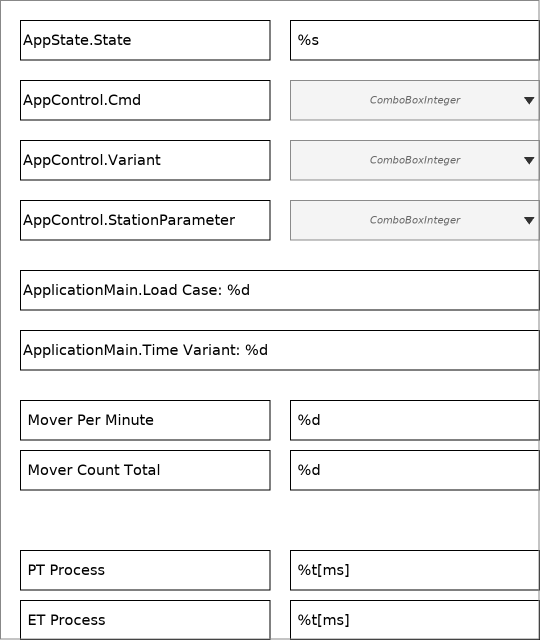
VISUALIZATION APP_CONTROL  // 540x640
    Rectangle (20,270 520x40), "ApplicationMain.Load Case: %d", text variable: GVL_APPLICATION.ApplicationMain._nLoadCase
        OnMouseClick: write the text variable via VisuDialogs.Numpad, min 0, max 2
    Rectangle (20,330 520x40), "ApplicationMain.Time Variant: %d", text variable: GVL_APPLICATION.ApplicationMain._nTimeVariant
        OnMouseClick: write the text variable via VisuDialogs.Numpad, min 0, max 100
    Rectangle (20,80 250x40), "AppControl.Cmd"
    ComboBoxInteger (290,80 250x40), variable: GVL_APPLICATION.AppControl.Cmd, text list: 'TL_E_INSTANCE_CMD'
    Rectangle (20,20 250x40), "AppState.State"
    Rectangle (290,20 250x40), "%s", text variable: GVL_APPLICATION.ApplicationMain._sAppState
    Rectangle (20,400 250x40), "Mover Per Minute", input disabled if: (MAIN.eInit = E_PROGRESS.PROGRESS_DONE)
    Rectangle (290,400 250x40), "%d", text variable: GVL_APPLICATION.AppInfo.MoverPerMinute, input disabled if: (MAIN.eInit = E_PROGRESS.PROGRESS_DONE)
    Rectangle (20,450 250x40), "Mover Count Total", input disabled if: (MAIN.eInit = E_PROGRESS.PROGRESS_DONE)
    Rectangle (290,450 250x40), "%d", text variable: GVL_APPLICATION.AppInfo.MoverTotal, input disabled if: (MAIN.eInit = E_PROGRESS.PROGRESS_DONE)
    Rectangle (20,600 250x40), "ET Process", input disabled if: (MAIN.eInit = E_PROGRESS.PROGRESS_DONE)
    Rectangle (290,600 250x40), "%t[ms]", text variable: GVL_APPLICATION.ApplicationMain._tonProcess[E_INSTANCE.INFEED].ET, input disabled if: (MAIN.eInit = E_PROGRESS.PROGRESS_DONE)
    Rectangle (20,550 250x40), "PT Process", input disabled if: (MAIN.eInit = E_PROGRESS.PROGRESS_DONE)
    Rectangle (290,550 250x40), "%t[ms]", text variable: GVL_APPLICATION.ApplicationMain._tProcess[E_INSTANCE.INFEED], input disabled if: (MAIN.eInit = E_PROGRESS.PROGRESS_DONE)
    Rectangle (20,140 250x40), "AppControl.Variant"
    ComboBoxInteger (290,140 250x40), variable: GVL_APPLICATION.AppControl.Variant, text list: 'TL_E_APP_VARIANT'
    Rectangle (20,200 250x40), "AppControl.StationParameter"
    ComboBoxInteger (290,200 250x40), variable: GVL_APPLICATION.AppControl.StationParameterVariant, text list: 'TL_E_STATION_PARAMETER_VARIANT'
END_VISUALIZATION

(* stored: Version 1.1.0.1
   Visu APP_CONTROL: Id {d7875bb1-1944-44dc-9a90-dd2ff6dca64b} *)
